INTERFACE ICollisionGroup

METHOD Disable : BOOL
VAR_INPUT
END_VAR
END_METHOD

METHOD Enable : BOOL
VAR_INPUT
END_VAR
END_METHOD

PROPERTY GroupRef : reference to AXES_GROUP_REF
GET
END_GET
END_PROPERTY

PROPERTY GroupState : CAGroupStatus
GET
END_GET
END_PROPERTY

METHOD Reset : BOOL
VAR_INPUT
END_VAR
END_METHOD

END_INTERFACE

(* stored: Version 1.1.0.1, ProductVersion 3.1.4024.11
   Itf ICollisionGroup: Id {a4a17a47-4830-427c-86d5-634057663097}
   Method Disable: Id {1571c256-d887-4291-b576-021e9805db7d}
   Method Enable: Id {2624ca75-8393-4480-808b-a75970c43af1}
   Property GroupRef: Id {764ba64e-bfd9-4632-b977-f2ca26e885b8}
   Get Get: Id {00d25a7c-3034-49b7-b381-f03d719a6f08}
   Property GroupState: Id {4a72ae6c-7470-4e2c-b03b-fb0755064c99}
   Get Get: Id {c9f590d7-83b8-495b-964c-f1b75d0f29ad}
   Method Reset: Id {fdebc938-e7b5-46db-a08c-2d5131d7e750} *)
